(* CODESYS project Winda2.project

Project tree, tasks and I/O mapping:
  Device : CODESYS Control Win V3, 3S - Smart Software Solutions GmbH, order no. 305021, version 3.5.8.10
    application Application
      libraries: Standard, * (System)
      task MainTask (cyclic, interval t#20ms, priority 1) calls PLC_PRG
      task VISU_TASK (cyclic, interval 100 ms, priority 31) calls VisuElems.Visu_Prg
      program PLC_PRG [CFC]
      visualisation Visualization
  libraries: VisuSymbols, 3.5.8.0 (System)
  text list GlobalTextList
*)

// Device/Application/PLC_PRG
PROGRAM PLC_PRG
VAR
	t1: TON;				// układ czasowy do szybkości windy
	zegar: BOOL;
	zmienna: TIME;
	rs1: RS;
	rs5: RS;
	przycisk_1: BOOL;
	przycisk_5: BOOL;
	winda_na_1: BOOL;
	winda_na_5: BOOL;
	winda_1: BOOL;
	winda_5: BOOL;
	licznik: WORD;
	C1: CTUD;
	rs2: RS;
	winda_4: BOOL;
	przycisk_2: BOOL;
	winda_na_2: BOOL;
	winda_2: BOOL;
	rs3: RS;
	winda_3: BOOL;
	przycisk_4: BOOL;
	winda_na_4: BOOL;
	przycisk_3: BOOL;
	winda_na_3: BOOL;
	rs4: RS;
END_VAR
VAR // added by the converter: edge detectors and wires of the graphical bodies
    _w1, _w2 : ANY;
END_VAR

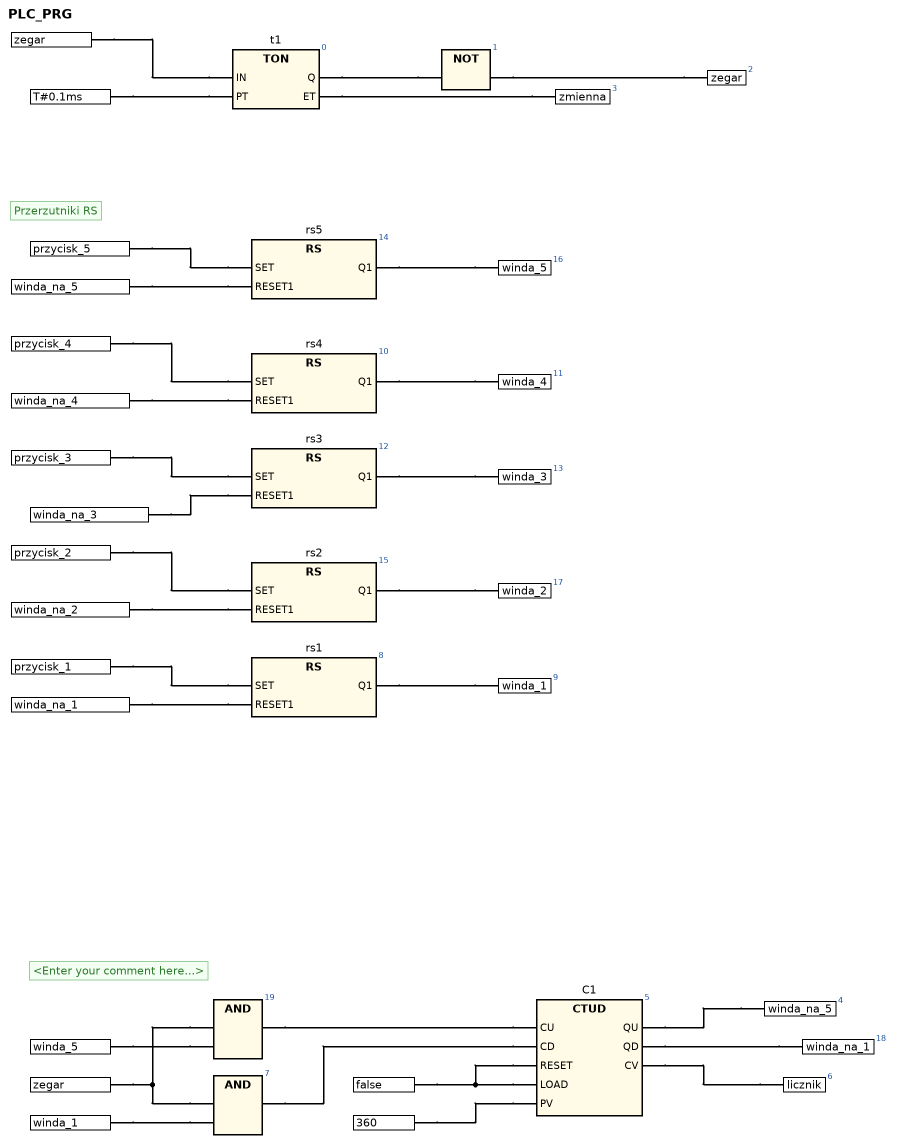
t1(IN := zegar, PT := T#0.1ms); // TON
zegar := NOT t1.Q;
zmienna := t1.ET;
winda_na_5 := C1.QU;
C1(CU := _w1, CD := _w2, RESET := false, LOAD := false, PV := 360); // CTUD
licznik := C1.CV;
_w2 := zegar AND winda_1;
rs1(SET := przycisk_1, RESET1 := winda_na_1); // RS
winda_1 := rs1.Q1;
rs4(SET := przycisk_4, RESET1 := winda_na_4); // RS
winda_4 := rs4.Q1;
rs3(SET := przycisk_3, RESET1 := winda_na_3); // RS
winda_3 := rs3.Q1;
// Przerzutniki RS
rs5(SET := przycisk_5, RESET1 := winda_na_5); // RS
rs2(SET := przycisk_2, RESET1 := winda_na_2); // RS
winda_5 := rs5.Q1;
winda_2 := rs2.Q1;
winda_na_1 := C1.QD;
// <Enter your comment here...>
_w1 := zegar AND winda_5;

END_PROGRAM

// Device/Application/Visualization
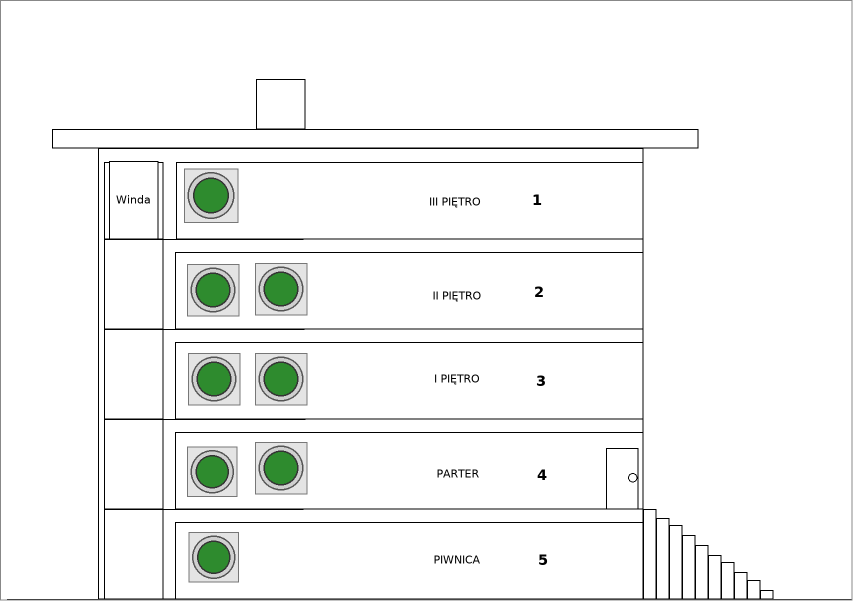
VISUALIZATION Visualization  // 853x601
    Rectangle (98,148 545x451)
    Rectangle (175,522 468x77)
    Rectangle (104,162 59x77)
    Rectangle (104,239 59x90)
    Rectangle (104,329 59x90)
    Rectangle (104,419 59x90)
    Rectangle (104,509 59x90)
    Rectangle (109,161 49x78), "Winda"
        p2738717112: PLC_PRG.licznik
    Rectangle (175,432 468x77)
    Rectangle (175,342 468x77)
    Rectangle (175,252 468x77)
    Rectangle (176,162 467x77)
    Rectangle (52,129 646x19)
    Rectangle (256,79 49x50)
    Line (652,599) (851,599)
    Rectangle (606,448 32x61)
    Rectangle (643,509 13x90)
    Rectangle (656,518 13x81)
    Rectangle (669,525 13x74)
    Rectangle (682,535 13x64)
    Rectangle (695,545 13x54)
    Rectangle (708,555 13x44)
    Rectangle (721,562 13x37)
    Rectangle (734,572 13x27)
    Rectangle (747,580 13x19)
    Rectangle (760,590 13x9)
    Line (7,599) (206,599)
    Line (104,509) (303,509)
    Line (106,419) (305,419)
    Line (105,329) (304,329)
    Line (104,239) (303,239)
    Ellipse (628,473 9x9)
    Label (382,545 150x30), "PIWNICA"
    Label (383,459 150x30), "PARTER"
    Label (382,364 150x30), "I PIĘTRO"
    Label (382,281 150x30), "II PIĘTRO"
    Label (380,187 150x30), "III PIĘTRO"
    PushSwitch (184,168 54x55), variable: PLC_PRG.przycisk_1, behaviour: TOGGLE, style: Switch-PushSwitch-Green
    PushSwitch (187,445 50x53), behaviour: TOGGLE, style: Switch-PushSwitch-Green
    PushSwitch (187,353 54x52), behaviour: TOGGLE, style: Switch-PushSwitch-Green
    PushSwitch (187,264 52x52), behaviour: TOGGLE, style: Switch-PushSwitch-Green
    PushSwitch (187,532 53x50), variable: PLC_PRG.przycisk_5, behaviour: TOGGLE, style: Switch-PushSwitch-Green
    PushSwitch (255,263 52x52), behaviour: TOGGLE, style: Switch-PushSwitch-Green
    PushSwitch (255,353 52x52), behaviour: TOGGLE, style: Switch-PushSwitch-Green
    PushSwitch (255,442 52x52), behaviour: TOGGLE, style: Switch-PushSwitch-Green
    Label (468,545 150x30), "5"
    Label (467,460 150x30), "4"
    Label (466,366 150x30), "3"
    Label (464,277 150x30), "2"
    Label (462,185 150x30), "1"
END_VISUALIZATION
